(* CODESYS project CleaningRobot.project

Project tree, tasks and I/O mapping:
  Device : AC801-0221-U0R0, Shenzhen Inovance Technology Co., Ltd., version 3.5.11.50
      settings: PersistentStartAdddr = 0; PersistentStartEndAddr = 5242879; Mode = 0
    application Application
      libraries: Standard, * (System); CmpHCCom, 1.1.0.1 (Inovance); HC_CommBus, 1.3.12.0 (Inovance); CallCFunction, 1.7.2 (Inovance); CmpHCCom, 1.1.0.1 (Inovance); CmpEventMgr, 3.5.8.0 (System); ISysTypes2, 3.5.0.0 (System); CmpApp, 3.5.11.0 (System); IOBlockHandle, 1.3.0.0 (Inovance); HC_OmronUtils, 1.5.4.0 (Inovance); VisuDialogs, * (System)
      task ETHERCAT_C (cyclic, interval 4000 µs, priority 0) calls ETHERCAT_C.EtherCAT_Task, PLC_PRG, AxisTest_PRG
      program PLC_PRG [ST]
      DifferentialMonitor
      Symbols
      function block EventCallbackFunBLock [ST]: EventCallback, FB_Exit, FB_Init
      trace Trace (task ETHERCAT_C): PLC_PRG.sMotionOutputs.dCmdPos[0], PLC_PRG.sMotionOutputs.dCmdPos[1], PLC_PRG.sMotionOutputs.dCmdPos[2], PLC_PRG.sMotionInputs.dFbPos[0], PLC_PRG.sMotionInputs.dFbPos[1], PLC_PRG.sMotionInputs.dFbPos[2], PLC_PRG.sMotionOutputs.dCmdSpace[0], PLC_PRG.sMotionOutputs.dCmdSpace[1], PLC_PRG.sMotionOutputs.dCmdSpace[2], PLC_PRG.sMotionInputs.dFbSpace[0]
      program AxisTest_PRG [ST]
    Network Configuration
      EtherCAT Config
    Resources List
    ConfigStorage
    HardWare Configuration
    Device Diagnosis
    SoftMotion General Axis Pool
    MODBUS_TCP : ModbusTCP本地从站, inovance, version 00.00.00.10
    HwConfiguratioinDevice : SystemConfig, Inovance, version 00.00.00.10
        settings: NetworkConfigArray.NetworkConfigArray.BusType = 10; NetworkConfigArray.NetworkConfigArray.RackSum = 1; NetworkConfigArray.NetworkConfigArray.HardwareConfigArray.HardwareConfigArray.RackNo = 1
    ETHERCAT_C : EtherCAT Master SoftMotion, 3S - Smart Software Solutions GmbH, version 3.5.11.10
        settings:  = 0; Autoconfig = 0; NetworkName = 'enp3s0'; SelectNetworkByName = TRUE; DisableTaskGeneration = True
      InoSV630N_机械臂3轴 : SV630_1Axis_03715, Inovance, order no. InoSV630N, version Revision=16#00010000
          settings: Number of Outputs = 6; Number of Inputs = 10; Number of Infos about Outputs = 6; Number of Infos about Inputs = 10; Physical Address of the Slave = 1003; AutoIncr Address of the Slave = 4294967294; StationAlias = 0; Sync.Length = 18; Sync.Length = 32; FMMU.Global Start Address = 16#02000025; FMMU.Length = 18; FMMU.Physical Start Address = 16#1800; FMMU.Access = 16#02; FMMU.Global Start Address = 16#01000040; FMMU.Length = 32; FMMU.Physical Start Address = 16#1C00; FMMU.Access = 16#01; FMMU.Global Start Address = 16#00080000; FMMU.StartBit = 2; FMMU.EndBit = 2; FMMU.Physical Start Address = 16#080D; FMMU.Access = 16#01; AutoUpdate = False; DC sync0 cycletime = 4000; DC sync1 cycletime = 4000; Number of SDO = 10; Homing method.Index = 16#6098; Homing method.Subindex = 16#00; Homing method.Value = 1; Homing method.Size = 8; Homing method.AbortIfError = FALSE; Homing method.JumpToLine = FALSE; Homing method.Line = 0; Homing method.CompleteAccess = FALSE; Actual Position Calculation Method.Index = 16#60E6; Actual Position Calculation Method.Subindex = 16#00; Actual Position Calculation Method.Value = 0; Actual Position Calculation Method.Size = 8; Actual Position Calculation Method.AbortIfError = FALSE; Actual Position Calculation Method.JumpToLine = FALSE;
            Actual Position Calculation Method.Line = 0; Actual Position Calculation Method.CompleteAccess = FALSE; Speed during search for switch.Index = 16#6099; Speed during search for switch.Subindex = 16#01; Speed during search for switch.Value = 436907; Speed during search for switch.Size = 32; Speed during search for switch.AbortIfError = FALSE; Speed during search for switch.JumpToLine = FALSE; Speed during search for switch.Line = 0; Speed during search for switch.CompleteAccess = FALSE; Homing acceleration.Index = 16#609A; Homing acceleration.Subindex = 16#00; Homing acceleration.Value = 43690666; Homing acceleration.Size = 32; Homing acceleration.AbortIfError = FALSE; Homing acceleration.JumpToLine = FALSE; Homing acceleration.Line = 0; Homing acceleration.CompleteAccess = FALSE; Speed during search for zero.Index = 16#6099; Speed during search for zero.Subindex = 16#02; Speed during search for zero.Value = 43691; Speed during search for zero.Size = 32; Speed during search for zero.AbortIfError = FALSE; Speed during search for zero.JumpToLine = FALSE; Speed during search for zero.Line = 0; Speed during search for zero.CompleteAccess = FALSE; Time of home searching.Index = 16#2005; Time of home searching.Subindex = 16#24; Time of home searching.Value = 50000; Time of home searching.Size = 16; Time of home searching.AbortIfError = FALSE; Time of home searching.JumpToLine = FALSE; Time of home searching.Line = 0; Time of home searching.CompleteAccess = FALSE; Positive torque limit value.Index = 16#60E0; Positive torque limit value.Subindex = 16#00; Positive torque limit value.Value = 3500; Positive torque limit value.Size = 16; Positive torque limit value.AbortIfError = FALSE; Positive torque limit value.JumpToLine = FALSE;
            Positive torque limit value.Line = 0; Positive torque limit value.CompleteAccess = FALSE; Negative torque limit value.Index = 16#60E1; Negative torque limit value.Subindex = 16#00; Negative torque limit value.Value = 3500; Negative torque limit value.Size = 16; Negative torque limit value.AbortIfError = FALSE; Negative torque limit value.JumpToLine = FALSE; Negative torque limit value.Line = 0; Negative torque limit value.CompleteAccess = FALSE; Max profile velocity.Index = 16#607F; Max profile velocity.Subindex = 16#00; Max profile velocity.Value = 26214400; Max profile velocity.Size = 32; Max profile velocity.AbortIfError = FALSE; Max profile velocity.JumpToLine = FALSE; Max profile velocity.Line = 0; Max profile velocity.CompleteAccess = FALSE; RxTxPdo.NumberofEntries = 6; RxTxPdo.Sm = 2; Controlword.Index = 16#6040; Controlword.SubIndex = 0; Controlword.Size = 16; Controlword.DependOnSlot = false; Controlword.DependOnSlotGroup = false; Target position.Index = 16#607A; Target position.SubIndex = 0; Target position.Size = 32; Target position.DependOnSlot = false; Target position.DependOnSlotGroup = false; Touch probe function.Index = 16#60B8; Touch probe function.SubIndex = 0; Touch probe function.Size = 16; Touch probe function.DependOnSlot = false; Touch probe function.DependOnSlotGroup = false; Physical outputs.Index = 16#60FE; Physical outputs.SubIndex = 1; Physical outputs.Size = 32; Physical outputs.DependOnSlot = false; Physical outputs.DependOnSlotGroup = false;
            Target velocity.Index = 16#60FF; Target velocity.SubIndex = 0; Target velocity.Size = 32; Target velocity.DependOnSlot = false; Target velocity.DependOnSlotGroup = false; Target torque.Index = 16#6071; Target torque.SubIndex = 0; Target torque.Size = 16; Target torque.DependOnSlot = false; Target torque.DependOnSlotGroup = false; RxTxPdo.Sm = -1; RxTxPdo.NumberofEntries = 10; RxTxPdo.Sm = 3; Error code.Index = 16#603F; Error code.SubIndex = 0; Error code.Size = 16; Error code.DependOnSlot = false; Error code.DependOnSlotGroup = false; Statusword.Index = 16#6041; Statusword.SubIndex = 0; Statusword.Size = 16; Statusword.DependOnSlot = false; Statusword.DependOnSlotGroup = false; Position actual value.Index = 16#6064; Position actual value.SubIndex = 0; Position actual value.Size = 32; Position actual value.DependOnSlot = false; Position actual value.DependOnSlotGroup = false; Torque actual value.Index = 16#6077; Torque actual value.SubIndex = 0; Torque actual value.Size = 16; Torque actual value.DependOnSlot = false; Torque actual value.DependOnSlotGroup = false; Following error actual value.Index = 16#60F4; Following error actual value.SubIndex = 0; Following error actual value.Size = 32; Following error actual value.DependOnSlot = false; Following error actual value.DependOnSlotGroup = false; Touch probe status.Index = 16#60B9; Touch probe status.SubIndex = 0;
            Touch probe status.Size = 16; Touch probe status.DependOnSlot = false; Touch probe status.DependOnSlotGroup = false; Touch probe pos1 pos value.Index = 16#60BA; Touch probe pos1 pos value.SubIndex = 0; Touch probe pos1 pos value.Size = 32; Touch probe pos1 pos value.DependOnSlot = false; Touch probe pos1 pos value.DependOnSlotGroup = false; Touch probe pos2 pos value.Index = 16#60BC; Touch probe pos2 pos value.SubIndex = 0; Touch probe pos2 pos value.Size = 32; Touch probe pos2 pos value.DependOnSlot = false; Touch probe pos2 pos value.DependOnSlotGroup = false; Digital inputs.Index = 16#60FD; Digital inputs.SubIndex = 0; Digital inputs.Size = 32; Digital inputs.DependOnSlot = false; Digital inputs.DependOnSlotGroup = false; Velocity actual value.Index = 16#606C; Velocity actual value.SubIndex = 0; Velocity actual value.Size = 32; Velocity actual value.DependOnSlot = false; Velocity actual value.DependOnSlotGroup = false; RxTxPdo.Sm = -1; Controlword.Name = 'Controlword'; Controlword.DataType = 'UINT'; Target position.Name = 'Target position'; Target position.DataType = 'DINT'; Touch probe function.Name = 'Touch probe function'; Touch probe function.DataType = 'UINT'; Physical outputs.Name = 'Physical outputs'; Physical outputs.DataType = 'UDINT'; Target velocity.Name = 'Target velocity'; Target velocity.DataType = 'DINT'; Target torque.Name = 'Target torque'; Target torque.DataType = 'INT'; Error code.Name = 'Error code'; Error code.DataType = 'UINT'; Statusword.Name = 'Statusword'; Statusword.DataType = 'UINT';
            Position actual value.Name = 'Position actual value'; Position actual value.DataType = 'DINT'; Torque actual value.Name = 'Torque actual value'; Torque actual value.DataType = 'INT'; Following error actual value.Name = 'Following error actual value'; Following error actual value.DataType = 'DINT'; Touch probe status.Name = 'Touch probe status'; Touch probe status.DataType = 'UINT'; Touch probe pos1 pos value.Name = 'Touch probe pos1 pos value'; Touch probe pos1 pos value.DataType = 'DINT'; Touch probe pos2 pos value.Name = 'Touch probe pos2 pos value'; Touch probe pos2 pos value.DataType = 'DINT'; Digital inputs.Name = 'Digital inputs'; Digital inputs.DataType = 'UDINT'; Velocity actual value.Name = 'Velocity actual value'; Velocity actual value.DataType = 'DINT'
          unmapped channels: Controlword, Target position, Touch probe function, Physical outputs, Target velocity, Target torque, Error code, Statusword, Position actual value, Torque actual value, Following error actual value, Touch probe status, Touch probe pos1 pos value, Touch probe pos2 pos value, Digital inputs, Velocity actual value
        机械臂3轴 : Axis, Inovance, order no. 0, version 1.0.0.0
            settings: wDriveID = 2; dwRatioTechUnitsDenom = 262144; fSWMaxVelocity = 1000; fSWMaxAcceleration = 10000; fSWMaxDeceleration = 10000; fSWMaxJerk = 100000; iEncoderType = 1; iAbsEncoderOption = 1; HomingMode = 10; ZeroSignal = 0; StartDirction = 1; EndDirection = 1; PosLimitMode = 0; NegLimitMode = 0; HomingVelocity = 10; HomingApproachVelocity = 2; HomingAcceleration = 100; HomingDeceleration = 100; HomingJerk = 0; HomeMaskDistance = 0; HomePositionOffset = 0; HomePushTime = 0; HomeCompensation = 0; HomeTimeout = 0; HomeCompensationVelocity = 1000; 4000 = 0; 4001 = 0; 4003 = true; 4004 = 3; 4005 = 0; 4006 = 1.666667; 4007 = 166.666666; 4008 = 0.166667; 4009 = 50000; 4010 = 3500; 4011 = 3500; 4012 = 100.000000; ScalingIncs = 16#40000; 6005 = 1; AdrOffset_8010 = 48;
              BitOffset_8010 = 0; BitLength_8010 = 16; Address_8010 = '%QW24'; Type_8010 = 'UINT'; AddressPointer_8010 = ADR(%QW24); AdrOffset_8020 = 52; BitOffset_8020 = 0; BitLength_8020 = 32; Address_8020 = '%QD13'; Type_8020 = 'DINT'; AddressPointer_8020 = ADR(%QD13); AdrOffset_8030 = 64; BitOffset_8030 = 0; BitLength_8030 = 32; Address_8030 = '%QD16'; Type_8030 = 'DINT'; AddressPointer_8030 = ADR(%QD16); AdrOffset_8040 = 68; BitOffset_8040 = 0; BitLength_8040 = 16; Address_8040 = '%QW34'; Type_8040 = 'INT'; AddressPointer_8040 = ADR(%QW34); AdrOffset_8050 = 4294967295; BitOffset_8050 = 0; BitLength_8050 = 0; Address_8050 = ''; Type_8050 = ''; AddressPointer_8050 = 0; AdrOffset_8060 = 56; BitOffset_8060 = 0; BitLength_8060 = 16; Address_8060 = '%QW28'; Type_8060 = 'UINT'; AddressPointer_8060 = ADR(%QW28); AdrOffset_8070 = 4294967295; BitOffset_8070 = 0; BitLength_8070 = 0; Address_8070 = ''; Type_8070 = '';
              AddressPointer_8070 = 0; AdrOffset_8080 = 4294967295; BitOffset_8080 = 0; BitLength_8080 = 0; Address_8080 = ''; Type_8080 = ''; AddressPointer_8080 = 0; AdrOffset_8090 = 60; BitOffset_8090 = 0; BitLength_8090 = 32; Address_8090 = '%QD15'; Type_8090 = 'UDINT'; AddressPointer_8090 = ADR(%QD15); AdrOffset_8100 = 4294967295; BitOffset_8100 = 0; BitLength_8100 = 0; Address_8100 = ''; Type_8100 = ''; AddressPointer_8100 = 0; AdrOffset_8510 = 74; BitOffset_8510 = 0; BitLength_8510 = 16; Address_8510 = '%IW37'; Type_8510 = 'UINT'; AddressPointer_8510 = ADR(%IW37); AdrOffset_8520 = 76; BitOffset_8520 = 0; BitLength_8520 = 32; Address_8520 = '%ID19'; Type_8520 = 'DINT'; AddressPointer_8520 = ADR(%ID19); AdrOffset_8530 = 104; BitOffset_8530 = 0; BitLength_8530 = 32; Address_8530 = '%ID26'; Type_8530 = 'DINT'; AddressPointer_8530 = ADR(%ID26); AdrOffset_8540 = 80; BitOffset_8540 = 0; BitLength_8540 = 16;
              Address_8540 = '%IW40'; Type_8540 = 'INT'; AddressPointer_8540 = ADR(%IW40); AdrOffset_8550 = 4294967295; BitOffset_8550 = 0; BitLength_8550 = 0; Address_8550 = ''; Type_8550 = ''; AddressPointer_8550 = 0; AdrOffset_8560 = 100; BitOffset_8560 = 0; BitLength_8560 = 32; Address_8560 = '%ID25'; Type_8560 = 'UDINT'; AddressPointer_8560 = ADR(%ID25); AdrOffset_8570 = 88; BitOffset_8570 = 0; BitLength_8570 = 16; Address_8570 = '%IW44'; Type_8570 = 'UINT'; AddressPointer_8570 = ADR(%IW44); AdrOffset_8580 = 92; BitOffset_8580 = 0; BitLength_8580 = 32; Address_8580 = '%ID23'; Type_8580 = 'DINT'; AddressPointer_8580 = ADR(%ID23); AdrOffset_8590 = 4294967295; BitOffset_8590 = 0; BitLength_8590 = 0; Address_8590 = ''; Type_8590 = ''; AddressPointer_8590 = 0; AdrOffset_8600 = 96; BitOffset_8600 = 0; BitLength_8600 = 32; Address_8600 = '%ID24'; Type_8600 = 'DINT'; AddressPointer_8600 = ADR(%ID24); AdrOffset_8600 = 4294967295;
              BitOffset_8600 = 0; BitLength_8600 = 0; Address_8610 = ''; Type_8610 = ''; AddressPointer_8610 = 0; AdrOffset_8620 = 72; BitOffset_8620 = 0; BitLength_8620 = 16; Address_8620 = '%IW36'; Type_8620 = 'UINT'; AddressPointer_8620 = ADR(%IW36); IsValid = True; IsHostHoming = False; PulseSelectIndex = 2
      InoSV630N_机械臂4轴 : SV630_1Axis_03715, Inovance, order no. InoSV630N, version Revision=16#00010000
          settings: Number of Outputs = 6; Number of Inputs = 10; Number of Infos about Outputs = 6; Number of Infos about Inputs = 10; Physical Address of the Slave = 1004; AutoIncr Address of the Slave = 4294967293; StationAlias = 0; Sync.Length = 18; Sync.Length = 32; FMMU.Global Start Address = 16#02000037; FMMU.Length = 18; FMMU.Physical Start Address = 16#1800; FMMU.Access = 16#02; FMMU.Global Start Address = 16#01000060; FMMU.Length = 32; FMMU.Physical Start Address = 16#1C00; FMMU.Access = 16#01; FMMU.Global Start Address = 16#00080000; FMMU.StartBit = 3; FMMU.EndBit = 3; FMMU.Physical Start Address = 16#080D; FMMU.Access = 16#01; AutoUpdate = False; DC sync0 cycletime = 4000; DC sync1 cycletime = 4000; Number of SDO = 10; Homing method.Index = 16#6098; Homing method.Subindex = 16#00; Homing method.Value = 1; Homing method.Size = 8; Homing method.AbortIfError = FALSE; Homing method.JumpToLine = FALSE; Homing method.Line = 0; Homing method.CompleteAccess = FALSE; Actual Position Calculation Method.Index = 16#60E6; Actual Position Calculation Method.Subindex = 16#00; Actual Position Calculation Method.Value = 0; Actual Position Calculation Method.Size = 8; Actual Position Calculation Method.AbortIfError = FALSE; Actual Position Calculation Method.JumpToLine = FALSE;
            Actual Position Calculation Method.Line = 0; Actual Position Calculation Method.CompleteAccess = FALSE; Speed during search for switch.Index = 16#6099; Speed during search for switch.Subindex = 16#01; Speed during search for switch.Value = 436907; Speed during search for switch.Size = 32; Speed during search for switch.AbortIfError = FALSE; Speed during search for switch.JumpToLine = FALSE; Speed during search for switch.Line = 0; Speed during search for switch.CompleteAccess = FALSE; Homing acceleration.Index = 16#609A; Homing acceleration.Subindex = 16#00; Homing acceleration.Value = 43690666; Homing acceleration.Size = 32; Homing acceleration.AbortIfError = FALSE; Homing acceleration.JumpToLine = FALSE; Homing acceleration.Line = 0; Homing acceleration.CompleteAccess = FALSE; Speed during search for zero.Index = 16#6099; Speed during search for zero.Subindex = 16#02; Speed during search for zero.Value = 43691; Speed during search for zero.Size = 32; Speed during search for zero.AbortIfError = FALSE; Speed during search for zero.JumpToLine = FALSE; Speed during search for zero.Line = 0; Speed during search for zero.CompleteAccess = FALSE; Time of home searching.Index = 16#2005; Time of home searching.Subindex = 16#24; Time of home searching.Value = 50000; Time of home searching.Size = 16; Time of home searching.AbortIfError = FALSE; Time of home searching.JumpToLine = FALSE; Time of home searching.Line = 0; Time of home searching.CompleteAccess = FALSE; Positive torque limit value.Index = 16#60E0; Positive torque limit value.Subindex = 16#00; Positive torque limit value.Value = 3500; Positive torque limit value.Size = 16; Positive torque limit value.AbortIfError = FALSE; Positive torque limit value.JumpToLine = FALSE;
            Positive torque limit value.Line = 0; Positive torque limit value.CompleteAccess = FALSE; Negative torque limit value.Index = 16#60E1; Negative torque limit value.Subindex = 16#00; Negative torque limit value.Value = 3500; Negative torque limit value.Size = 16; Negative torque limit value.AbortIfError = FALSE; Negative torque limit value.JumpToLine = FALSE; Negative torque limit value.Line = 0; Negative torque limit value.CompleteAccess = FALSE; Max profile velocity.Index = 16#607F; Max profile velocity.Subindex = 16#00; Max profile velocity.Value = 26214400; Max profile velocity.Size = 32; Max profile velocity.AbortIfError = FALSE; Max profile velocity.JumpToLine = FALSE; Max profile velocity.Line = 0; Max profile velocity.CompleteAccess = FALSE; RxTxPdo.NumberofEntries = 6; RxTxPdo.Sm = 2; Controlword.Index = 16#6040; Controlword.SubIndex = 0; Controlword.Size = 16; Controlword.DependOnSlot = false; Controlword.DependOnSlotGroup = false; Target position.Index = 16#607A; Target position.SubIndex = 0; Target position.Size = 32; Target position.DependOnSlot = false; Target position.DependOnSlotGroup = false; Touch probe function.Index = 16#60B8; Touch probe function.SubIndex = 0; Touch probe function.Size = 16; Touch probe function.DependOnSlot = false; Touch probe function.DependOnSlotGroup = false; Physical outputs.Index = 16#60FE; Physical outputs.SubIndex = 1; Physical outputs.Size = 32; Physical outputs.DependOnSlot = false; Physical outputs.DependOnSlotGroup = false;
            Target velocity.Index = 16#60FF; Target velocity.SubIndex = 0; Target velocity.Size = 32; Target velocity.DependOnSlot = false; Target velocity.DependOnSlotGroup = false; Target torque.Index = 16#6071; Target torque.SubIndex = 0; Target torque.Size = 16; Target torque.DependOnSlot = false; Target torque.DependOnSlotGroup = false; RxTxPdo.Sm = -1; RxTxPdo.NumberofEntries = 10; RxTxPdo.Sm = 3; Error code.Index = 16#603F; Error code.SubIndex = 0; Error code.Size = 16; Error code.DependOnSlot = false; Error code.DependOnSlotGroup = false; Statusword.Index = 16#6041; Statusword.SubIndex = 0; Statusword.Size = 16; Statusword.DependOnSlot = false; Statusword.DependOnSlotGroup = false; Position actual value.Index = 16#6064; Position actual value.SubIndex = 0; Position actual value.Size = 32; Position actual value.DependOnSlot = false; Position actual value.DependOnSlotGroup = false; Torque actual value.Index = 16#6077; Torque actual value.SubIndex = 0; Torque actual value.Size = 16; Torque actual value.DependOnSlot = false; Torque actual value.DependOnSlotGroup = false; Following error actual value.Index = 16#60F4; Following error actual value.SubIndex = 0; Following error actual value.Size = 32; Following error actual value.DependOnSlot = false; Following error actual value.DependOnSlotGroup = false; Touch probe status.Index = 16#60B9; Touch probe status.SubIndex = 0;
            Touch probe status.Size = 16; Touch probe status.DependOnSlot = false; Touch probe status.DependOnSlotGroup = false; Touch probe pos1 pos value.Index = 16#60BA; Touch probe pos1 pos value.SubIndex = 0; Touch probe pos1 pos value.Size = 32; Touch probe pos1 pos value.DependOnSlot = false; Touch probe pos1 pos value.DependOnSlotGroup = false; Touch probe pos2 pos value.Index = 16#60BC; Touch probe pos2 pos value.SubIndex = 0; Touch probe pos2 pos value.Size = 32; Touch probe pos2 pos value.DependOnSlot = false; Touch probe pos2 pos value.DependOnSlotGroup = false; Digital inputs.Index = 16#60FD; Digital inputs.SubIndex = 0; Digital inputs.Size = 32; Digital inputs.DependOnSlot = false; Digital inputs.DependOnSlotGroup = false; Velocity actual value.Index = 16#606C; Velocity actual value.SubIndex = 0; Velocity actual value.Size = 32; Velocity actual value.DependOnSlot = false; Velocity actual value.DependOnSlotGroup = false; RxTxPdo.Sm = -1; Controlword.Name = 'Controlword'; Controlword.DataType = 'UINT'; Target position.Name = 'Target position'; Target position.DataType = 'DINT'; Touch probe function.Name = 'Touch probe function'; Touch probe function.DataType = 'UINT'; Physical outputs.Name = 'Physical outputs'; Physical outputs.DataType = 'UDINT'; Target velocity.Name = 'Target velocity'; Target velocity.DataType = 'DINT'; Target torque.Name = 'Target torque'; Target torque.DataType = 'INT'; Error code.Name = 'Error code'; Error code.DataType = 'UINT'; Statusword.Name = 'Statusword'; Statusword.DataType = 'UINT';
            Position actual value.Name = 'Position actual value'; Position actual value.DataType = 'DINT'; Torque actual value.Name = 'Torque actual value'; Torque actual value.DataType = 'INT'; Following error actual value.Name = 'Following error actual value'; Following error actual value.DataType = 'DINT'; Touch probe status.Name = 'Touch probe status'; Touch probe status.DataType = 'UINT'; Touch probe pos1 pos value.Name = 'Touch probe pos1 pos value'; Touch probe pos1 pos value.DataType = 'DINT'; Touch probe pos2 pos value.Name = 'Touch probe pos2 pos value'; Touch probe pos2 pos value.DataType = 'DINT'; Digital inputs.Name = 'Digital inputs'; Digital inputs.DataType = 'UDINT'; Velocity actual value.Name = 'Velocity actual value'; Velocity actual value.DataType = 'DINT'
          unmapped channels: Controlword, Target position, Touch probe function, Physical outputs, Target velocity, Target torque, Error code, Statusword, Position actual value, Torque actual value, Following error actual value, Touch probe status, Touch probe pos1 pos value, Touch probe pos2 pos value, Digital inputs, Velocity actual value
        机械臂4轴 : Axis, Inovance, order no. 0, version 1.0.0.0
            settings: wDriveID = 3; dwRatioTechUnitsDenom = 262144; fSWMaxVelocity = 1000; fSWMaxAcceleration = 10000; fSWMaxDeceleration = 10000; fSWMaxJerk = 100000; iEncoderType = 1; iAbsEncoderOption = 1; HomingMode = 10; ZeroSignal = 0; StartDirction = 1; EndDirection = 1; PosLimitMode = 0; NegLimitMode = 0; HomingVelocity = 10; HomingApproachVelocity = 2; HomingAcceleration = 100; HomingDeceleration = 100; HomingJerk = 0; HomeMaskDistance = 0; HomePositionOffset = 0; HomePushTime = 0; HomeCompensation = 0; HomeTimeout = 0; HomeCompensationVelocity = 1000; 4000 = 0; 4001 = 0; 4003 = true; 4004 = 3; 4005 = 0; 4006 = 1.666667; 4007 = 166.666666; 4008 = 0.166667; 4009 = 50000; 4010 = 3500; 4011 = 3500; 4012 = 100.000000; ScalingIncs = 16#40000; 6005 = 1; AdrOffset_8010 = 72;
              BitOffset_8010 = 0; BitLength_8010 = 16; Address_8010 = '%QW36'; Type_8010 = 'UINT'; AddressPointer_8010 = ADR(%QW36); AdrOffset_8020 = 76; BitOffset_8020 = 0; BitLength_8020 = 32; Address_8020 = '%QD19'; Type_8020 = 'DINT'; AddressPointer_8020 = ADR(%QD19); AdrOffset_8030 = 88; BitOffset_8030 = 0; BitLength_8030 = 32; Address_8030 = '%QD22'; Type_8030 = 'DINT'; AddressPointer_8030 = ADR(%QD22); AdrOffset_8040 = 92; BitOffset_8040 = 0; BitLength_8040 = 16; Address_8040 = '%QW46'; Type_8040 = 'INT'; AddressPointer_8040 = ADR(%QW46); AdrOffset_8050 = 4294967295; BitOffset_8050 = 0; BitLength_8050 = 0; Address_8050 = ''; Type_8050 = ''; AddressPointer_8050 = 0; AdrOffset_8060 = 80; BitOffset_8060 = 0; BitLength_8060 = 16; Address_8060 = '%QW40'; Type_8060 = 'UINT'; AddressPointer_8060 = ADR(%QW40); AdrOffset_8070 = 4294967295; BitOffset_8070 = 0; BitLength_8070 = 0; Address_8070 = ''; Type_8070 = '';
              AddressPointer_8070 = 0; AdrOffset_8080 = 4294967295; BitOffset_8080 = 0; BitLength_8080 = 0; Address_8080 = ''; Type_8080 = ''; AddressPointer_8080 = 0; AdrOffset_8090 = 84; BitOffset_8090 = 0; BitLength_8090 = 32; Address_8090 = '%QD21'; Type_8090 = 'UDINT'; AddressPointer_8090 = ADR(%QD21); AdrOffset_8100 = 4294967295; BitOffset_8100 = 0; BitLength_8100 = 0; Address_8100 = ''; Type_8100 = ''; AddressPointer_8100 = 0; AdrOffset_8510 = 110; BitOffset_8510 = 0; BitLength_8510 = 16; Address_8510 = '%IW55'; Type_8510 = 'UINT'; AddressPointer_8510 = ADR(%IW55); AdrOffset_8520 = 112; BitOffset_8520 = 0; BitLength_8520 = 32; Address_8520 = '%ID28'; Type_8520 = 'DINT'; AddressPointer_8520 = ADR(%ID28); AdrOffset_8530 = 140; BitOffset_8530 = 0; BitLength_8530 = 32; Address_8530 = '%ID35'; Type_8530 = 'DINT'; AddressPointer_8530 = ADR(%ID35); AdrOffset_8540 = 116; BitOffset_8540 = 0; BitLength_8540 = 16;
              Address_8540 = '%IW58'; Type_8540 = 'INT'; AddressPointer_8540 = ADR(%IW58); AdrOffset_8550 = 4294967295; BitOffset_8550 = 0; BitLength_8550 = 0; Address_8550 = ''; Type_8550 = ''; AddressPointer_8550 = 0; AdrOffset_8560 = 136; BitOffset_8560 = 0; BitLength_8560 = 32; Address_8560 = '%ID34'; Type_8560 = 'UDINT'; AddressPointer_8560 = ADR(%ID34); AdrOffset_8570 = 124; BitOffset_8570 = 0; BitLength_8570 = 16; Address_8570 = '%IW62'; Type_8570 = 'UINT'; AddressPointer_8570 = ADR(%IW62); AdrOffset_8580 = 128; BitOffset_8580 = 0; BitLength_8580 = 32; Address_8580 = '%ID32'; Type_8580 = 'DINT'; AddressPointer_8580 = ADR(%ID32); AdrOffset_8590 = 4294967295; BitOffset_8590 = 0; BitLength_8590 = 0; Address_8590 = ''; Type_8590 = ''; AddressPointer_8590 = 0; AdrOffset_8600 = 132; BitOffset_8600 = 0; BitLength_8600 = 32; Address_8600 = '%ID33'; Type_8600 = 'DINT'; AddressPointer_8600 = ADR(%ID33); AdrOffset_8600 = 4294967295;
              BitOffset_8600 = 0; BitLength_8600 = 0; Address_8610 = ''; Type_8610 = ''; AddressPointer_8610 = 0; AdrOffset_8620 = 108; BitOffset_8620 = 0; BitLength_8620 = 16; Address_8620 = '%IW54'; Type_8620 = 'UINT'; AddressPointer_8620 = ADR(%IW54); IsValid = True; IsHostHoming = False; PulseSelectIndex = 2
      InoSV630N_机械臂1轴 : SV630_1Axis_03715, Inovance, order no. InoSV630N, version Revision=16#00010000
          settings: Number of Outputs = 7; Number of Inputs = 10; Number of Infos about Outputs = 7; Number of Infos about Inputs = 10; Physical Address of the Slave = 1001; StationAlias = 0; Sync.Length = 19; Sync.Length = 32; FMMU.Global Start Address = 16#02000000; FMMU.Length = 19; FMMU.Physical Start Address = 16#1800; FMMU.Access = 16#02; FMMU.Global Start Address = 16#01000000; FMMU.Length = 32; FMMU.Physical Start Address = 16#1C00; FMMU.Access = 16#01; FMMU.Global Start Address = 16#00080000; FMMU.Physical Start Address = 16#080D; FMMU.Access = 16#01; AutoUpdate = False; DC sync0 cycletime = 4000; DC sync1 cycletime = 4000; Number of SDO = 10; Homing method.Index = 16#6098; Homing method.Subindex = 16#00; Homing method.Value = 1; Homing method.Size = 8; Homing method.AbortIfError = FALSE; Homing method.JumpToLine = FALSE; Homing method.Line = 0; Homing method.CompleteAccess = False; Actual Position Calculation Method.Index = 16#60E6; Actual Position Calculation Method.Subindex = 16#00; Actual Position Calculation Method.Value = 0; Actual Position Calculation Method.Size = 8; Actual Position Calculation Method.AbortIfError = FALSE; Actual Position Calculation Method.JumpToLine = FALSE; Actual Position Calculation Method.Line = 0; Actual Position Calculation Method.CompleteAccess = False; Speed during search for switch.Index = 16#6099;
            Speed during search for switch.Subindex = 16#01; Speed during search for switch.Value = 436907; Speed during search for switch.Size = 32; Speed during search for switch.AbortIfError = FALSE; Speed during search for switch.JumpToLine = FALSE; Speed during search for switch.Line = 0; Speed during search for switch.CompleteAccess = False; Homing acceleration.Index = 16#609A; Homing acceleration.Subindex = 16#00; Homing acceleration.Value = 43690666; Homing acceleration.Size = 32; Homing acceleration.AbortIfError = FALSE; Homing acceleration.JumpToLine = FALSE; Homing acceleration.Line = 0; Homing acceleration.CompleteAccess = False; Speed during search for zero.Index = 16#6099; Speed during search for zero.Subindex = 16#02; Speed during search for zero.Value = 43691; Speed during search for zero.Size = 32; Speed during search for zero.AbortIfError = FALSE; Speed during search for zero.JumpToLine = FALSE; Speed during search for zero.Line = 0; Speed during search for zero.CompleteAccess = False; Time of home searching.Index = 16#2005; Time of home searching.Subindex = 16#24; Time of home searching.Value = 50000; Time of home searching.Size = 16; Time of home searching.AbortIfError = FALSE; Time of home searching.JumpToLine = FALSE; Time of home searching.Line = 0; Time of home searching.CompleteAccess = False; Positive torque limit value.Index = 16#60E0; Positive torque limit value.Subindex = 16#00; Positive torque limit value.Value = 3500; Positive torque limit value.Size = 16; Positive torque limit value.AbortIfError = FALSE; Positive torque limit value.JumpToLine = FALSE; Positive torque limit value.Line = 0; Positive torque limit value.CompleteAccess = False; Negative torque limit value.Index = 16#60E1;
            Negative torque limit value.Subindex = 16#00; Negative torque limit value.Value = 3500; Negative torque limit value.Size = 16; Negative torque limit value.AbortIfError = FALSE; Negative torque limit value.JumpToLine = FALSE; Negative torque limit value.Line = 0; Negative torque limit value.CompleteAccess = False; Max profile velocity.Index = 16#607F; Max profile velocity.Subindex = 16#00; Max profile velocity.Value = 26214400; Max profile velocity.Size = 32; Max profile velocity.AbortIfError = FALSE; Max profile velocity.JumpToLine = FALSE; Max profile velocity.Line = 0; Max profile velocity.CompleteAccess = False; RxTxPdo.NumberofEntries = 7; RxTxPdo.Sm = 2; RxTxPdo.DependOnSlot = False; RxTxPdo.DependOnSlotGroup = False; RxTxPdo.OverwrittenByModule = False; Exclude = [16#1701,16#1702,16#1703,16#1704,16#1705]; Controlword.Index = 16#6040; Controlword.SubIndex = 0; Controlword.Size = 16; Controlword.Offset = 0; Controlword.DependOnSlot = False; Controlword.DependOnSlotGroup = False; Target position.Index = 16#607A; Target position.SubIndex = 0; Target position.Size = 32; Target position.Offset = 0; Target position.DependOnSlot = False; Target position.DependOnSlotGroup = False; Touch probe function.Index = 16#60B8; Touch probe function.SubIndex = 0; Touch probe function.Size = 16; Touch probe function.Offset = 0; Touch probe function.DependOnSlot = False; Touch probe function.DependOnSlotGroup = False; Physical outputs.Index = 16#60FE;
            Physical outputs.SubIndex = 1; Physical outputs.Size = 32; Physical outputs.Offset = 0; Physical outputs.DependOnSlot = False; Physical outputs.DependOnSlotGroup = False; Target velocity.Index = 16#60FF; Target velocity.SubIndex = 0; Target velocity.Size = 32; Target velocity.Offset = 0; Target velocity.DependOnSlot = False; Target velocity.DependOnSlotGroup = False; Modes of operation.Index = 16#6060; Modes of operation.SubIndex = 0; Modes of operation.Size = 8; Modes of operation.Offset = 0; Modes of operation.DependOnSlot = False; Modes of operation.DependOnSlotGroup = False; Target torque.Index = 16#6071; Target torque.SubIndex = 0; Target torque.Size = 16; Target torque.Offset = 0; Target torque.DependOnSlot = False; Target torque.DependOnSlotGroup = False; RxTxPdo.Sm = -1; RxTxPdo.NumberofEntries = 10; RxTxPdo.Sm = 3; Error code.Index = 16#603F; Error code.SubIndex = 0; Error code.Size = 16; Error code.DependOnSlot = false; Error code.DependOnSlotGroup = false; Statusword.Index = 16#6041; Statusword.SubIndex = 0; Statusword.Size = 16; Statusword.DependOnSlot = false; Statusword.DependOnSlotGroup = false; Position actual value.Index = 16#6064; Position actual value.SubIndex = 0; Position actual value.Size = 32; Position actual value.DependOnSlot = false;
            Position actual value.DependOnSlotGroup = false; Torque actual value.Index = 16#6077; Torque actual value.SubIndex = 0; Torque actual value.Size = 16; Torque actual value.DependOnSlot = false; Torque actual value.DependOnSlotGroup = false; Following error actual value.Index = 16#60F4; Following error actual value.SubIndex = 0; Following error actual value.Size = 32; Following error actual value.DependOnSlot = false; Following error actual value.DependOnSlotGroup = false; Touch probe status.Index = 16#60B9; Touch probe status.SubIndex = 0; Touch probe status.Size = 16; Touch probe status.DependOnSlot = false; Touch probe status.DependOnSlotGroup = false; Touch probe pos1 pos value.Index = 16#60BA; Touch probe pos1 pos value.SubIndex = 0; Touch probe pos1 pos value.Size = 32; Touch probe pos1 pos value.DependOnSlot = false; Touch probe pos1 pos value.DependOnSlotGroup = false; Touch probe pos2 pos value.Index = 16#60BC; Touch probe pos2 pos value.SubIndex = 0; Touch probe pos2 pos value.Size = 32; Touch probe pos2 pos value.DependOnSlot = false; Touch probe pos2 pos value.DependOnSlotGroup = false; Digital inputs.Index = 16#60FD; Digital inputs.SubIndex = 0; Digital inputs.Size = 32; Digital inputs.DependOnSlot = false; Digital inputs.DependOnSlotGroup = false; Velocity actual value.Index = 16#606C; Velocity actual value.SubIndex = 0; Velocity actual value.Size = 32; Velocity actual value.DependOnSlot = false; Velocity actual value.DependOnSlotGroup = false; RxTxPdo.Sm = -1; Controlword.Name = 'Controlword'; Controlword.DataType = 'UINT'; Controlword.Default = '';
            Controlword.Comment = ''; Target position.Name = 'Target position'; Target position.DataType = 'DINT'; Target position.Default = ''; Target position.Comment = ''; Touch probe function.Name = 'Touch probe function'; Touch probe function.DataType = 'UINT'; Touch probe function.Default = ''; Touch probe function.Comment = ''; Physical outputs.Name = 'Physical outputs'; Physical outputs.DataType = 'UDINT'; Physical outputs.Default = ''; Physical outputs.Comment = ''; Target velocity.Name = 'Target velocity'; Target velocity.DataType = 'DINT'; Target velocity.Default = ''; Target velocity.Comment = ''; Modes of operation.Name = 'Modes of operation'; Modes of operation.DataType = 'SINT'; Modes of operation.Default = ''; Modes of operation.Comment = ''; Target torque.Name = 'Target torque'; Target torque.DataType = 'INT'; Target torque.Default = ''; Target torque.Comment = ''; Error code.Name = 'Error code'; Error code.DataType = 'UINT'; Statusword.Name = 'Statusword'; Statusword.DataType = 'UINT'; Position actual value.Name = 'Position actual value'; Position actual value.DataType = 'DINT'; Torque actual value.Name = 'Torque actual value'; Torque actual value.DataType = 'INT'; Following error actual value.Name = 'Following error actual value'; Following error actual value.DataType = 'DINT'; Touch probe status.Name = 'Touch probe status'; Touch probe status.DataType = 'UINT'; Touch probe pos1 pos value.Name = 'Touch probe pos1 pos value'; Touch probe pos1 pos value.DataType = 'DINT'; Touch probe pos2 pos value.Name = 'Touch probe pos2 pos value';
            Touch probe pos2 pos value.DataType = 'DINT'; Digital inputs.Name = 'Digital inputs'; Digital inputs.DataType = 'UDINT'; Velocity actual value.Name = 'Velocity actual value'; Velocity actual value.DataType = 'DINT'
          input  Application.AxisTest_PRG.adFbPos[0] : DINT  // Position actual value
          unmapped channels: Controlword, Target position, Touch probe function, Physical outputs, Target velocity, Modes of operation, Target torque, Error code, Statusword, Torque actual value, Following error actual value, Touch probe status, Touch probe pos1 pos value, Touch probe pos2 pos value, Digital inputs, Velocity actual value
        机械臂1轴 : Axis, Inovance, order no. 0, version 1.0.0.0
            settings: wDriveID = 0; dwRatioTechUnitsDenom = 262144; fSWMaxVelocity = 1000; fSWMaxAcceleration = 10000; fSWMaxDeceleration = 10000; fSWMaxJerk = 100000; iEncoderType = 1; iAbsEncoderOption = 1; HomingMode = 10; ZeroSignal = 0; StartDirction = 1; EndDirection = 1; PosLimitMode = 0; NegLimitMode = 0; HomingVelocity = 10; HomingApproachVelocity = 2; HomingAcceleration = 100; HomingDeceleration = 100; HomingJerk = 0; HomeMaskDistance = 0; HomePositionOffset = 0; HomePushTime = 0; HomeCompensation = 0; HomeTimeout = 0; HomeCompensationVelocity = 1000; 4000 = 0; 4001 = 0; 4003 = true; 4004 = 3; 4005 = 0; 4006 = 1.666667; 4007 = 166.666666; 4008 = 0.166667; 4009 = 50000; 4010 = 3500; 4011 = 3500; 4012 = 100.000000; ScalingIncs = 16#40000; 6005 = 1; AdrOffset_8010 = 0;
              BitOffset_8010 = 0; BitLength_8010 = 16; Address_8010 = '%QW0'; Type_8010 = 'UINT'; AddressPointer_8010 = ADR(%QW0); AdrOffset_8020 = 4; BitOffset_8020 = 0; BitLength_8020 = 32; Address_8020 = '%QD1'; Type_8020 = 'DINT'; AddressPointer_8020 = ADR(%QD1); AdrOffset_8030 = 16; BitOffset_8030 = 0; BitLength_8030 = 32; Address_8030 = '%QD4'; Type_8030 = 'DINT'; AddressPointer_8030 = ADR(%QD4); AdrOffset_8040 = 22; BitOffset_8040 = 0; BitLength_8040 = 16; Address_8040 = '%QW11'; Type_8040 = 'INT'; AddressPointer_8040 = ADR(%QW11); AdrOffset_8050 = 20; BitOffset_8050 = 0; BitLength_8050 = 8; Address_8050 = '%QB20'; Type_8050 = 'SINT'; AddressPointer_8050 = ADR(%QB20); AdrOffset_8060 = 8; BitOffset_8060 = 0; BitLength_8060 = 16; Address_8060 = '%QW4'; Type_8060 = 'UINT'; AddressPointer_8060 = ADR(%QW4); AdrOffset_8070 = 4294967295; BitOffset_8070 = 0; BitLength_8070 = 0; Address_8070 = ''; Type_8070 = '';
              AddressPointer_8070 = 0; AdrOffset_8080 = 4294967295; BitOffset_8080 = 0; BitLength_8080 = 0; Address_8080 = ''; Type_8080 = ''; AddressPointer_8080 = 0; AdrOffset_8090 = 12; BitOffset_8090 = 0; BitLength_8090 = 32; Address_8090 = '%QD3'; Type_8090 = 'UDINT'; AddressPointer_8090 = ADR(%QD3); AdrOffset_8100 = 4294967295; BitOffset_8100 = 0; BitLength_8100 = 0; Address_8100 = ''; Type_8100 = ''; AddressPointer_8100 = 0; AdrOffset_8510 = 2; BitOffset_8510 = 0; BitLength_8510 = 16; Address_8510 = '%IW1'; Type_8510 = 'UINT'; AddressPointer_8510 = ADR(%IW1); AdrOffset_8520 = 0; BitOffset_8520 = 0; BitLength_8520 = 32; Address_8520 = 'AxisTest_PRG.adFbPos[0]'; Type_8520 = 'DINT'; AddressPointer_8520 = ADR(AxisTest_PRG.adFbPos[0]); AdrOffset_8530 = 32; BitOffset_8530 = 0; BitLength_8530 = 32; Address_8530 = '%ID8'; Type_8530 = 'DINT'; AddressPointer_8530 = ADR(%ID8); AdrOffset_8540 = 8; BitOffset_8540 = 0; BitLength_8540 = 16;
              Address_8540 = '%IW4'; Type_8540 = 'INT'; AddressPointer_8540 = ADR(%IW4); AdrOffset_8550 = 4294967295; BitOffset_8550 = 0; BitLength_8550 = 0; Address_8550 = ''; Type_8550 = ''; AddressPointer_8550 = 0; AdrOffset_8560 = 28; BitOffset_8560 = 0; BitLength_8560 = 32; Address_8560 = '%ID7'; Type_8560 = 'UDINT'; AddressPointer_8560 = ADR(%ID7); AdrOffset_8570 = 16; BitOffset_8570 = 0; BitLength_8570 = 16; Address_8570 = '%IW8'; Type_8570 = 'UINT'; AddressPointer_8570 = ADR(%IW8); AdrOffset_8580 = 20; BitOffset_8580 = 0; BitLength_8580 = 32; Address_8580 = '%ID5'; Type_8580 = 'DINT'; AddressPointer_8580 = ADR(%ID5); AdrOffset_8590 = 4294967295; BitOffset_8590 = 0; BitLength_8590 = 0; Address_8590 = ''; Type_8590 = ''; AddressPointer_8590 = 0; AdrOffset_8600 = 24; BitOffset_8600 = 0; BitLength_8600 = 32; Address_8600 = '%ID6'; Type_8600 = 'DINT'; AddressPointer_8600 = ADR(%ID6); AdrOffset_8600 = 4294967295;
              BitOffset_8600 = 0; BitLength_8600 = 0; Address_8610 = ''; Type_8610 = ''; AddressPointer_8610 = 0; AdrOffset_8620 = 0; BitOffset_8620 = 0; BitLength_8620 = 16; Address_8620 = '%IW0'; Type_8620 = 'UINT'; AddressPointer_8620 = ADR(%IW0); Automatic Mapping = True; IsValid = True; IsHostHoming = False; PulseSelectIndex = 2
      InoSV630N_机械臂2轴 : SV630_1Axis_03715, Inovance, order no. InoSV630N, version Revision=16#00010000
          settings: Number of Outputs = 6; Number of Inputs = 10; Number of Infos about Outputs = 6; Number of Infos about Inputs = 10; Physical Address of the Slave = 1002; AutoIncr Address of the Slave = 4294967295; StationAlias = 0; Sync.Length = 18; Sync.Length = 32; FMMU.Global Start Address = 16#02000013; FMMU.Length = 18; FMMU.Physical Start Address = 16#1800; FMMU.Access = 16#02; FMMU.Global Start Address = 16#01000020; FMMU.Length = 32; FMMU.Physical Start Address = 16#1C00; FMMU.Access = 16#01; FMMU.Global Start Address = 16#00080000; FMMU.StartBit = 1; FMMU.EndBit = 1; FMMU.Physical Start Address = 16#080D; FMMU.Access = 16#01; AutoUpdate = False; DC sync0 cycletime = 4000; DC sync1 cycletime = 4000; Number of SDO = 10; Homing method.Index = 16#6098; Homing method.Subindex = 16#00; Homing method.Value = 1; Homing method.Size = 8; Homing method.AbortIfError = FALSE; Homing method.JumpToLine = FALSE; Homing method.Line = 0; Homing method.CompleteAccess = FALSE; Actual Position Calculation Method.Index = 16#60E6; Actual Position Calculation Method.Subindex = 16#00; Actual Position Calculation Method.Value = 0; Actual Position Calculation Method.Size = 8; Actual Position Calculation Method.AbortIfError = FALSE; Actual Position Calculation Method.JumpToLine = FALSE;
            Actual Position Calculation Method.Line = 0; Actual Position Calculation Method.CompleteAccess = FALSE; Speed during search for switch.Index = 16#6099; Speed during search for switch.Subindex = 16#01; Speed during search for switch.Value = 436907; Speed during search for switch.Size = 32; Speed during search for switch.AbortIfError = FALSE; Speed during search for switch.JumpToLine = FALSE; Speed during search for switch.Line = 0; Speed during search for switch.CompleteAccess = FALSE; Homing acceleration.Index = 16#609A; Homing acceleration.Subindex = 16#00; Homing acceleration.Value = 43690666; Homing acceleration.Size = 32; Homing acceleration.AbortIfError = FALSE; Homing acceleration.JumpToLine = FALSE; Homing acceleration.Line = 0; Homing acceleration.CompleteAccess = FALSE; Speed during search for zero.Index = 16#6099; Speed during search for zero.Subindex = 16#02; Speed during search for zero.Value = 43691; Speed during search for zero.Size = 32; Speed during search for zero.AbortIfError = FALSE; Speed during search for zero.JumpToLine = FALSE; Speed during search for zero.Line = 0; Speed during search for zero.CompleteAccess = FALSE; Time of home searching.Index = 16#2005; Time of home searching.Subindex = 16#24; Time of home searching.Value = 50000; Time of home searching.Size = 16; Time of home searching.AbortIfError = FALSE; Time of home searching.JumpToLine = FALSE; Time of home searching.Line = 0; Time of home searching.CompleteAccess = FALSE; Positive torque limit value.Index = 16#60E0; Positive torque limit value.Subindex = 16#00; Positive torque limit value.Value = 3500; Positive torque limit value.Size = 16; Positive torque limit value.AbortIfError = FALSE; Positive torque limit value.JumpToLine = FALSE;
            Positive torque limit value.Line = 0; Positive torque limit value.CompleteAccess = FALSE; Negative torque limit value.Index = 16#60E1; Negative torque limit value.Subindex = 16#00; Negative torque limit value.Value = 3500; Negative torque limit value.Size = 16; Negative torque limit value.AbortIfError = FALSE; Negative torque limit value.JumpToLine = FALSE; Negative torque limit value.Line = 0; Negative torque limit value.CompleteAccess = FALSE; Max profile velocity.Index = 16#607F; Max profile velocity.Subindex = 16#00; Max profile velocity.Value = 26214400; Max profile velocity.Size = 32; Max profile velocity.AbortIfError = FALSE; Max profile velocity.JumpToLine = FALSE; Max profile velocity.Line = 0; Max profile velocity.CompleteAccess = FALSE; RxTxPdo.NumberofEntries = 6; RxTxPdo.Sm = 2; Controlword.Index = 16#6040; Controlword.SubIndex = 0; Controlword.Size = 16; Controlword.DependOnSlot = false; Controlword.DependOnSlotGroup = false; Target position.Index = 16#607A; Target position.SubIndex = 0; Target position.Size = 32; Target position.DependOnSlot = false; Target position.DependOnSlotGroup = false; Touch probe function.Index = 16#60B8; Touch probe function.SubIndex = 0; Touch probe function.Size = 16; Touch probe function.DependOnSlot = false; Touch probe function.DependOnSlotGroup = false; Physical outputs.Index = 16#60FE; Physical outputs.SubIndex = 1; Physical outputs.Size = 32; Physical outputs.DependOnSlot = false; Physical outputs.DependOnSlotGroup = false;
            Target velocity.Index = 16#60FF; Target velocity.SubIndex = 0; Target velocity.Size = 32; Target velocity.DependOnSlot = false; Target velocity.DependOnSlotGroup = false; Target torque.Index = 16#6071; Target torque.SubIndex = 0; Target torque.Size = 16; Target torque.DependOnSlot = false; Target torque.DependOnSlotGroup = false; RxTxPdo.Sm = -1; RxTxPdo.NumberofEntries = 10; RxTxPdo.Sm = 3; Error code.Index = 16#603F; Error code.SubIndex = 0; Error code.Size = 16; Error code.DependOnSlot = false; Error code.DependOnSlotGroup = false; Statusword.Index = 16#6041; Statusword.SubIndex = 0; Statusword.Size = 16; Statusword.DependOnSlot = false; Statusword.DependOnSlotGroup = false; Position actual value.Index = 16#6064; Position actual value.SubIndex = 0; Position actual value.Size = 32; Position actual value.DependOnSlot = false; Position actual value.DependOnSlotGroup = false; Torque actual value.Index = 16#6077; Torque actual value.SubIndex = 0; Torque actual value.Size = 16; Torque actual value.DependOnSlot = false; Torque actual value.DependOnSlotGroup = false; Following error actual value.Index = 16#60F4; Following error actual value.SubIndex = 0; Following error actual value.Size = 32; Following error actual value.DependOnSlot = false; Following error actual value.DependOnSlotGroup = false; Touch probe status.Index = 16#60B9; Touch probe status.SubIndex = 0;
            Touch probe status.Size = 16; Touch probe status.DependOnSlot = false; Touch probe status.DependOnSlotGroup = false; Touch probe pos1 pos value.Index = 16#60BA; Touch probe pos1 pos value.SubIndex = 0; Touch probe pos1 pos value.Size = 32; Touch probe pos1 pos value.DependOnSlot = false; Touch probe pos1 pos value.DependOnSlotGroup = false; Touch probe pos2 pos value.Index = 16#60BC; Touch probe pos2 pos value.SubIndex = 0; Touch probe pos2 pos value.Size = 32; Touch probe pos2 pos value.DependOnSlot = false; Touch probe pos2 pos value.DependOnSlotGroup = false; Digital inputs.Index = 16#60FD; Digital inputs.SubIndex = 0; Digital inputs.Size = 32; Digital inputs.DependOnSlot = false; Digital inputs.DependOnSlotGroup = false; Velocity actual value.Index = 16#606C; Velocity actual value.SubIndex = 0; Velocity actual value.Size = 32; Velocity actual value.DependOnSlot = false; Velocity actual value.DependOnSlotGroup = false; RxTxPdo.Sm = -1; Controlword.Name = 'Controlword'; Controlword.DataType = 'UINT'; Target position.Name = 'Target position'; Target position.DataType = 'DINT'; Touch probe function.Name = 'Touch probe function'; Touch probe function.DataType = 'UINT'; Physical outputs.Name = 'Physical outputs'; Physical outputs.DataType = 'UDINT'; Target velocity.Name = 'Target velocity'; Target velocity.DataType = 'DINT'; Target torque.Name = 'Target torque'; Target torque.DataType = 'INT'; Error code.Name = 'Error code'; Error code.DataType = 'UINT'; Statusword.Name = 'Statusword'; Statusword.DataType = 'UINT';
            Position actual value.Name = 'Position actual value'; Position actual value.DataType = 'DINT'; Torque actual value.Name = 'Torque actual value'; Torque actual value.DataType = 'INT'; Following error actual value.Name = 'Following error actual value'; Following error actual value.DataType = 'DINT'; Touch probe status.Name = 'Touch probe status'; Touch probe status.DataType = 'UINT'; Touch probe pos1 pos value.Name = 'Touch probe pos1 pos value'; Touch probe pos1 pos value.DataType = 'DINT'; Touch probe pos2 pos value.Name = 'Touch probe pos2 pos value'; Touch probe pos2 pos value.DataType = 'DINT'; Digital inputs.Name = 'Digital inputs'; Digital inputs.DataType = 'UDINT'; Velocity actual value.Name = 'Velocity actual value'; Velocity actual value.DataType = 'DINT'
          unmapped channels: Controlword, Target position, Touch probe function, Physical outputs, Target velocity, Target torque, Error code, Statusword, Position actual value, Torque actual value, Following error actual value, Touch probe status, Touch probe pos1 pos value, Touch probe pos2 pos value, Digital inputs, Velocity actual value
        机械臂2轴 : Axis, Inovance, order no. 0, version 1.0.0.0
            settings: dwRatioTechUnitsDenom = 262144; fSWMaxVelocity = 1000; fSWMaxAcceleration = 10000; fSWMaxDeceleration = 10000; fSWMaxJerk = 100000; iEncoderType = 1; iAbsEncoderOption = 1; HomingMode = 10; ZeroSignal = 0; StartDirction = 1; EndDirection = 1; PosLimitMode = 0; NegLimitMode = 0; HomingVelocity = 10; HomingApproachVelocity = 2; HomingAcceleration = 100; HomingDeceleration = 100; HomingJerk = 0; HomeMaskDistance = 0; HomePositionOffset = 0; HomePushTime = 0; HomeCompensation = 0; HomeTimeout = 0; HomeCompensationVelocity = 1000; 4000 = 0; 4001 = 0; 4003 = true; 4004 = 3; 4005 = 0; 4006 = 1.666667; 4007 = 166.666666; 4008 = 0.166667; 4009 = 50000; 4010 = 3500; 4011 = 3500; 4012 = 100.000000; ScalingIncs = 16#40000; 6005 = 1; AdrOffset_8010 = 24; BitOffset_8010 = 0;
              BitLength_8010 = 16; Address_8010 = '%QW12'; Type_8010 = 'UINT'; AddressPointer_8010 = ADR(%QW12); AdrOffset_8020 = 28; BitOffset_8020 = 0; BitLength_8020 = 32; Address_8020 = '%QD7'; Type_8020 = 'DINT'; AddressPointer_8020 = ADR(%QD7); AdrOffset_8030 = 40; BitOffset_8030 = 0; BitLength_8030 = 32; Address_8030 = '%QD10'; Type_8030 = 'DINT'; AddressPointer_8030 = ADR(%QD10); AdrOffset_8040 = 44; BitOffset_8040 = 0; BitLength_8040 = 16; Address_8040 = '%QW22'; Type_8040 = 'INT'; AddressPointer_8040 = ADR(%QW22); AdrOffset_8050 = 4294967295; BitOffset_8050 = 0; BitLength_8050 = 0; Address_8050 = ''; Type_8050 = ''; AddressPointer_8050 = 0; AdrOffset_8060 = 32; BitOffset_8060 = 0; BitLength_8060 = 16; Address_8060 = '%QW16'; Type_8060 = 'UINT'; AddressPointer_8060 = ADR(%QW16); AdrOffset_8070 = 4294967295; BitOffset_8070 = 0; BitLength_8070 = 0; Address_8070 = ''; Type_8070 = ''; AddressPointer_8070 = 0;
              AdrOffset_8080 = 4294967295; BitOffset_8080 = 0; BitLength_8080 = 0; Address_8080 = ''; Type_8080 = ''; AddressPointer_8080 = 0; AdrOffset_8090 = 36; BitOffset_8090 = 0; BitLength_8090 = 32; Address_8090 = '%QD9'; Type_8090 = 'UDINT'; AddressPointer_8090 = ADR(%QD9); AdrOffset_8100 = 4294967295; BitOffset_8100 = 0; BitLength_8100 = 0; Address_8100 = ''; Type_8100 = ''; AddressPointer_8100 = 0; AdrOffset_8510 = 38; BitOffset_8510 = 0; BitLength_8510 = 16; Address_8510 = '%IW19'; Type_8510 = 'UINT'; AddressPointer_8510 = ADR(%IW19); AdrOffset_8520 = 40; BitOffset_8520 = 0; BitLength_8520 = 32; Address_8520 = '%ID10'; Type_8520 = 'DINT'; AddressPointer_8520 = ADR(%ID10); AdrOffset_8530 = 68; BitOffset_8530 = 0; BitLength_8530 = 32; Address_8530 = '%ID17'; Type_8530 = 'DINT'; AddressPointer_8530 = ADR(%ID17); AdrOffset_8540 = 44; BitOffset_8540 = 0; BitLength_8540 = 16; Address_8540 = '%IW22';
              Type_8540 = 'INT'; AddressPointer_8540 = ADR(%IW22); AdrOffset_8550 = 4294967295; BitOffset_8550 = 0; BitLength_8550 = 0; Address_8550 = ''; Type_8550 = ''; AddressPointer_8550 = 0; AdrOffset_8560 = 64; BitOffset_8560 = 0; BitLength_8560 = 32; Address_8560 = '%ID16'; Type_8560 = 'UDINT'; AddressPointer_8560 = ADR(%ID16); AdrOffset_8570 = 52; BitOffset_8570 = 0; BitLength_8570 = 16; Address_8570 = '%IW26'; Type_8570 = 'UINT'; AddressPointer_8570 = ADR(%IW26); AdrOffset_8580 = 56; BitOffset_8580 = 0; BitLength_8580 = 32; Address_8580 = '%ID14'; Type_8580 = 'DINT'; AddressPointer_8580 = ADR(%ID14); AdrOffset_8590 = 4294967295; BitOffset_8590 = 0; BitLength_8590 = 0; Address_8590 = ''; Type_8590 = ''; AddressPointer_8590 = 0; AdrOffset_8600 = 60; BitOffset_8600 = 0; BitLength_8600 = 32; Address_8600 = '%ID15'; Type_8600 = 'DINT'; AddressPointer_8600 = ADR(%ID15); AdrOffset_8600 = 4294967295; BitOffset_8600 = 0;
              BitLength_8600 = 0; Address_8610 = ''; Type_8610 = ''; AddressPointer_8610 = 0; AdrOffset_8620 = 36; BitOffset_8620 = 0; BitLength_8620 = 16; Address_8620 = '%IW18'; Type_8620 = 'UINT'; AddressPointer_8620 = ADR(%IW18); IsValid = True; IsHostHoming = False; PulseSelectIndex = 2
  libraries: VisuSymbols, 3.5.10.0 (System)
  text list GlobalTextList
  data type MYIOBLOCK
  data type MOTION_INPUTS
  data type MOTION_OUTPUTS
  data type MOTION_EXTRADATA
*)

// MYIOBLOCK
{attribute 'pack_mode' := '1'}
TYPE MYIOBLOCK :
STRUCT
	ptr      : POINTER TO BYTE;           // inputs or outputs, and this ptr must be the first one
	len      : UINT;                      // size of the inputs or outpus
	name     : STRING(125);               // inputs or outputs name
END_STRUCT
END_TYPE

// MOTION_INPUTS
{attribute 'pack_mode' := '1'}
TYPE MOTION_INPUTS :
STRUCT
	iStatus   : INT;
	iServoErr : INT;
	dFbPos 	  : ARRAY[0..8] OF LREAL;
	dFbVel 	  : ARRAY[0..8] OF LREAL;
	dFbAcc 	  : ARRAY[0..8] OF LREAL;
	dFbSpace  : ARRAY[0..8] OF LREAL;
END_STRUCT
END_TYPE

// MOTION_OUTPUTS
{attribute 'pack_mode' := '1'}
TYPE MOTION_OUTPUTS :
STRUCT
	iRobStatus : INT;
	iErrorNum  : INT;
	dCmdPos  : ARRAY[0..8] OF LREAL;
	dCmdVel  : ARRAY[0..8] OF LREAL;
	dCmdAcc  : ARRAY[0..8] OF LREAL;
	dCmdSpace  : ARRAY[0..8] OF LREAL;
END_STRUCT
END_TYPE

// MOTION_EXTRADATA
{attribute 'pack_mode' := '1'}
TYPE MOTION_EXTRADATA :
STRUCT
	iPlanMode : INT;	// 0-手动, 1-自动
	bIsJoint  : BOOL;
	iAxisNum  : INT;
	bDir      : BOOL;
	dPos	  : ARRAY[0..8] OF LREAL;
END_STRUCT
END_TYPE

// Device/Application/PLC_PRG
PROGRAM PLC_PRG
VAR
	// 结构体
	sMotionInputs          	: MOTION_INPUTS;
	sMotionOutputs         	: MOTION_OUTPUTS;
	sMotionBlockInputs     	: MYIOBLOCK;
	sMotionBlockOutputs   	: MYIOBLOCK;
	sMotionExtraData       	: MOTION_EXTRADATA;
	sMotionPlanData        	: MOTION_EXTRADATA;
	
	// 函数
	fpMotionPlanCall       	: IOBlockCall;
	fpMotionMoveCall   	   	: IOBlockProcess;
	fpEventFB              	: EventCallbackFunBLock;
	
	// 变量
	xEnable                	: BOOL := TRUE;
	xPlanErr               	: BOOL;
	iPlanErrID             	: INT;
	xMoveErr               	: BOOL;
	iMoveErrID             	: INT;	
	
	iCounter			   	: INT := 0;
	bFirstRun			   	: BOOL := TRUE;
	bPlanMode			   	: INT :=0;
	bMotionPlanRun		  	: BOOL := FALSE;
	
	bSetHome		  		: BOOL := FALSE;
	adDisPos			   	: ARRAY[0..8] OF LREAL;
	adHomePos			   	: ARRAY[0..8] OF LREAL := [0.0, -90.0, 180.0, 90, 1, 1, 1, 1, 1];
	adZeroPos			   	: ARRAY[0..8] OF LREAL;
	
	aiAxisPnum			   	: ARRAY[0..8] OF DINT := [1, 1, 1, 1, 1, 1, 1, 1, 1];
	adGearRatio			   	: ARRAY[0..8] OF LREAL := [15.0, 15.0, 15.0, 15.0, 1.0, 1.0, 1.0, 1.0, 1.0];
	adPulseEqu			   	: ARRAY[0..8] OF LREAL;
	aiCcmdac			   	: ARRAY[0..8] OF LREAL;
	aiCfbPos     			: ARRAY[0..3] OF LREAL;
	
	bEnable	    			: BOOL := FALSE;
	apAxis      			: ARRAY[0..3] OF POINTER TO AXIS_REF_SM3;//定义轴
	apMC_Power  			: ARRAY[0..3] OF MC_Power;
END_VAR

sMotionBlockInputs.name      := 'motioninputs';
sMotionBlockInputs.len       := SIZEOF(sMotionInputs);
sMotionBlockInputs.ptr       := ADR(sMotionInputs);

sMotionBlockOutputs.name     := 'motionoutputs';
sMotionBlockOutputs.len      := SIZEOF(sMotionOutputs);
sMotionBlockOutputs.ptr      := ADR(sMotionOutputs);

// 第一次执行
IF bFirstRun THEN
	
	FOR iCounter:=0 TO 8 BY 1 DO
		adPulseEqu[iCounter] := aiAxisPnum[iCounter] * adGearRatio[iCounter] / 360.0;
	END_FOR
	
	// sMotionPlanData.iPlanMode := 1;	// 手动模式
	sMotionPlanData.iAxisNum := 0;
	sMotionPlanData.bDir := TRUE;
	sMotionPlanData.bIsJoint := TRUE;
	sMotionPlanData.dPos[0] := 0.0; sMotionPlanData.dPos[1] := -90.0; sMotionPlanData.dPos[2] := 180.0;
	sMotionPlanData.dPos[3] := 90.0; sMotionPlanData.dPos[4] := 0.0; sMotionPlanData.dPos[5] := 0.0;
	
	sMotionOutputs.dCmdPos[0] := 0.0; sMotionOutputs.dCmdPos[1] := -90.0; sMotionOutputs.dCmdPos[2] := 180.0;
	sMotionOutputs.dCmdPos[3] := 90.0; sMotionOutputs.dCmdPos[4] := 0.0; sMotionOutputs.dCmdPos[5] := 0.0;
	
	sMotionInputs.dFbPos[0] := 0.0; sMotionInputs.dFbPos[1] := -90.0; sMotionInputs.dFbPos[2] := 180.0;
	sMotionInputs.dFbPos[3] := 90.0; sMotionInputs.dFbPos[4] := 0.0; sMotionInputs.dFbPos[5] := 0.0;
	
	apAxis[0] := ADR(机械臂1轴);
	apAxis[1] := ADR(机械臂2轴);
	apAxis[2] := ADR(机械臂3轴);
	apAxis[3] := ADR(机械臂4轴);
	
	bFirstRun := FALSE;
END_IF

IF bSetHome = TRUE THEN
	FOR iCounter:=0 TO 8 BY 1 DO
		adDisPos[iCounter] := adDisPos[iCounter] + sMotionInputs.dFbPos[iCounter] - adHomePos[iCounter];
		adZeroPos[iCounter] := adDisPos[iCounter] - adHomePos[iCounter];
	END_FOR
	bSetHome := FALSE;
END_IF

// 运动完成
IF (sMotionOutputs.iRobStatus = 3) OR (sMotionOutputs.iRobStatus = 0) THEN
	sMotionPlanData.iPlanMode := 0;	// 空闲
	bMotionPlanRun := TRUE;
END_IF

IF bMotionPlanRun = TRUE THEN
	fpMotionPlanCall(
		xEnable               := xEnable,
		dwID                  := 1001,
		strFunName            := 'MotionPlan',
		pExtraData            := ADR(sMotionPlanData),
		xError                => xPlanErr, 
		eErrorID              => iPlanErrID
		);
	bMotionPlanRun := FALSE;
END_IF

fpMotionMoveCall(
	xEnable               := xEnable,
	dwID                  := 1001,
	pInputs               := ADR(sMotionBlockInputs),
	pOutputs              := ADR(sMotionBlockOutputs),
	strFunName            := 'MotionMove',
	pExtraData            := ADR(sMotionExtraData),
	xError                => xMoveErr,
	eErrorID              => iMoveErrID
	);

FOR iCounter:=0 TO 8 BY 1 DO
	aiCcmdac[iCounter] := (sMotionOutputs.dCmdPos[iCounter] + adZeroPos[iCounter]) * adPulseEqu[iCounter];
// 	sMotionInputs.dFbPos[iCounter] := (plus / adPulseEqu[iCounter]) - adZeroPos[iCounter];
	IF sMotionOutputs.dCmdPos[iCounter] <> 0 THEN
		apAxis[iCounter]^.fSetPosition := aiCcmdac[iCounter];
	END_IF
END_FOR

// IF sMotionOutputs.iRobStatus <> 1 THEN
// 	sMotionInputs.dFbPos[0] := sMotionOutputs.dCmdPos[0]; sMotionInputs.dFbPos[1] := sMotionOutputs.dCmdPos[1]; sMotionInputs.dFbPos[2] := sMotionOutputs.dCmdPos[2];
// 	sMotionInputs.dFbPos[3] := sMotionOutputs.dCmdPos[3]; sMotionInputs.dFbPos[4] := sMotionOutputs.dCmdPos[4]; sMotionInputs.dFbPos[5] := sMotionOutputs.dCmdPos[5];
// END_IF

aiCfbPos[0] := apAxis[0]^.fActPosition;
aiCfbPos[1] := apAxis[1]^.fActPosition;
aiCfbPos[2] := apAxis[2]^.fActPosition;
aiCfbPos[3] := apAxis[3]^.fActPosition;

sMotionInputs.dFbPos[0] := (apAxis[0]^.fActPosition / adPulseEqu[0]) - adZeroPos[0];
sMotionInputs.dFbPos[1] := (apAxis[1]^.fActPosition / adPulseEqu[1]) - adZeroPos[1];
sMotionInputs.dFbPos[2] := (apAxis[2]^.fActPosition / adPulseEqu[2]) - adZeroPos[2];
sMotionInputs.dFbPos[3] := (apAxis[3]^.fActPosition / adPulseEqu[3]) - adZeroPos[3];

END_PROGRAM

// Device/Application/EventCallbackFunBLock
FUNCTION_BLOCK EventCallbackFunBLock IMPLEMENTS ICmpEventCallback
VAR_INPUT
END_VAR
VAR_OUTPUT
END_VAR
VAR
	hEventStart			: RTS_IEC_HANDLE;
	hEventStop 			: RTS_IEC_HANDLE;
	hInterfaceStart 	: RTS_IEC_HANDLE;
	hInterfaceStop 		: RTS_IEC_HANDLE;
	ItfEventCallback 	: ICmpEventCallback;
	Result 				: UDINT;
END_VAR

METHOD EventCallback : UDINT
VAR_INPUT
	pEventParam : POINTER TO EventParam;
END_VAR
VAR
	pfIOBlockCall : IOBlockCall;
END_VAR
(* For every registered event this functions is called, because the function block
   implements ICmpEventCallback. *)

(* Save the stop Reason in a global variable *)
IF pEventParam^.EventId = EVT_StartDone THEN
	pfIOBlockCall(xEnable:=TRUE, dwID:=1001, strFunName:='ExampleInitialize', pExtraData:=(*custom data*));
ELSIF pEventParam^.EventId = EVT_PrepareStop THEN
	pfIOBlockCall(xEnable:=TRUE, dwID:=1001, strFunName:='ExampleRelease', pExtraData:=(*custom data*));
END_IF
END_METHOD

METHOD FB_Exit : BOOL
VAR_INPUT
	bInCopyCode: BOOL;
END_VAR
VAR
END_VAR
(* Unregister and close both Events *)
EventUnregisterCallback(hEventStart, hInterfaceStart);
EventUnregisterCallback(hEventStop, hInterfaceStop);

Result := EventClose2(hEventStart);
Result := EventClose2(hEventStop);
END_METHOD

METHOD FB_Init : BOOL
VAR_INPUT
	bInitRetains: BOOL;
	bInCopyCode: BOOL;	
END_VAR
VAR
END_VAR
ItfEventCallback := THIS^;

(* Open an Event which listens to the start Event *)
hEventStart := EventOpen(EVT_StartDone, CMPID_CmpApp, Result);
(* Open an Event which listens to the stop Event *)
hEventStop := EventOpen(EVT_PrepareStop, CMPID_CmpApp, Result);

(* Register the Interface Callback functions to the event. *)
hInterfaceStart := EventRegisterCallback(hEventStart, ItfEventCallback, Result);	
hInterfaceStop := EventRegisterCallback(hEventStop, ItfEventCallback, Result);
END_METHOD

END_FUNCTION_BLOCK

// Device/Application/AxisTest_PRG
PROGRAM AxisTest_PRG
VAR
	iCounter	: INT := 0;
	bMoveStatus	: INT := 0;
	iVel		: INT := 10;
	bFirstRun	: BOOL := TRUE;
	bEnable	    : BOOL := FALSE;
	bForward	: BOOL := FALSE;
	bBackward	: BOOL := FALSE;
	bMoveStart	: BOOL := FALSE;
	
	bSinMove    : BOOL := FALSE;
	dSinAmpl	: LREAL := 0.01;  // 振幅
	lSinFreq    : LREAL := 1;	  // 频率
	lSinFreqStep: LREAL := 3.0;
	lResult     : LREAL;
	adFbPos     : ARRAY[0..3] OF DINT;
	
	apMC_Jog    : ARRAY[0..3] OF MC_Jog;
	apMC_Power  : ARRAY[0..3] OF MC_Power;
	apAxis      : ARRAY[0..3] OF POINTER TO AXIS_REF_SM3;//定义轴
	apMC_MoveAbsolute : ARRAY[0..3] OF MC_MoveAbsolute;	//功能块声明
	apMC_Reset  : ARRAY[0..3] OF MC_Reset;
END_VAR

IF bFirstRun THEN
	apAxis[0] := ADR(机械臂1轴);
	apAxis[1] := ADR(机械臂2轴);
	apAxis[2] := ADR(机械臂3轴);
	apAxis[3] := ADR(机械臂4轴);
	bForward := TRUE;
	bBackward := TRUE;
	bFirstRun := FALSE;
END_IF

CASE bMoveStatus OF
	0 :
		bForward := TRUE;
		bBackward := FALSE;
	1 :
		bForward := FALSE;
		bBackward := TRUE;
	2 :
		bForward := FALSE;
		bBackward := FALSE;
END_CASE

FOR iCounter:=0 TO 3 BY 1 DO
	apMC_Power[iCounter](
		Axis:= apAxis[iCounter]^,
		Enable:= TRUE,
		bRegulatorOn:= bEnable,
		bDriveStart:= TRUE,
		Status=> , 
		bRegulatorRealState=> , 
		bDriveStartRealState=> , 
		Busy=> , 
		Error=> , 
		ErrorID=> );
END_FOR


// apMC_Power[0](
// 	Axis:= apAxis[0]^,
// 	Enable:= TRUE,
// 	bRegulatorOn:= bEnable,
// 	bDriveStart:= TRUE,
// 	Status=> , 
// 	bRegulatorRealState=> , 
// 	bDriveStartRealState=> , 
// 	Busy=> , 
// 	Error=> , 
// 	ErrorID=> );


IF bMoveStart = TRUE THEN
	FOR iCounter:=0 TO 3 BY 1 DO
		apMC_Jog[iCounter](
			Axis:= apAxis[iCounter]^, 
			JogForward:= bForward, 
			JogBackward:= bBackward, 
			Velocity:= iVel, 
			Acceleration:= 100, 
			Deceleration:= 100, 
			Jerk:=, 
			Busy=> , 
			CommandAborted=> , 
			Error=> , 
			ErrorId=> );
	END_FOR	
END_IF

IF bSinMove THEN
	lResult := SIN(0.0005 * lSinFreq) * dSinAmpl;
	lSinFreq := lSinFreq + lSinFreqStep;
	
	apAxis[0]^.fSetPosition := apAxis[0]^.fSetPosition + lResult;		//插补下发	
	apAxis[1]^.fSetPosition := apAxis[1]^.fSetPosition + lResult;
	apAxis[2]^.fSetPosition := apAxis[2]^.fSetPosition + lResult;
	apAxis[3]^.fSetPosition := apAxis[3]^.fSetPosition + lResult;
END_IF

// adFbPos[0] := apAxis[0]^.fActPosition;
// adFbPos[1] := apAxis[1]^.fActPosition;
// adFbPos[2] := apAxis[2]^.fActPosition;
// adFbPos[3] := apAxis[3]^.fActPosition;

FOR iCounter:=0 TO 3 BY 1 DO
	apMC_Reset[iCounter](Axis:=apAxis[iCounter]^, Execute:= , Done=> , Busy=> , Error=> , ErrorID=> );
END_FOR

END_PROGRAM
